FUNCTION_BLOCK MUX_UINT (* See MUX_ANY *)
  (* Standard: 61131-3 *)
  (* Version 0.0, 2004-12-15, JHC, Rockwell Automation, Converted from SRC format. *)
  (* Compiler header: package fb.rt.plc.select; *)
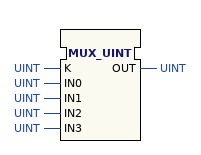
  VAR_INPUT
    K : UINT;
    IN0 : UINT;
    IN1 : UINT;
    IN2 : UINT;
    IN3 : UINT;
  END_VAR
  VAR_OUTPUT
    OUT : UINT;
  END_VAR
END_FUNCTION_BLOCK
